FUNCTION_BLOCK EL4022
VAR
	_io : EL4xx2_Data;
	{attribute addProperty Name "WcState"}
	_wcState : WcStateBase;
	{attribute addProperty Name "Info data"}
	_infoData : InfoDataAds;
END_VAR

PROPERTY IO : REFERENCE TO EL4xx2_Data
GET
IO REF= _io;
END_GET
END_PROPERTY

PROPERTY WcState : REFERENCE TO WcStateBase
GET
WcState REF= _wcState;
END_GET
END_PROPERTY

END_FUNCTION_BLOCK

(* stored: Version 1.1.0.1, ProductVersion 3.1.4024.9
   POU EL4022: Id {1b3ef903-af88-091c-136e-26ecfe771854}, SpecialFunc None
   Property IO: Id {a0b95b55-09a4-0152-3df3-824f0d2ba7e9}
   Get Get: Id {8bffe68b-612c-0026-1f95-9dc4692c7ccd}
   Property WcState: Id {309d7bda-da9f-0ff9-250e-c64d230a21f0}
   Get Get: Id {040ee16d-6524-0140-22fd-d24bfd8b03ba} *)
